// TwinCAT 3 PLC project PlcHammer
// Title: PlcHammer
// Company: TcOpenGroup
// ProjectVersion: 0.0.0.1
// ProgramVersion: 3.1.4023.0
// libraries:
//   Tc2_Math, * (Beckhoff Automation GmbH)
//   Tc2_Standard, * (Beckhoff Automation GmbH)
//   Tc2_System, * (Beckhoff Automation GmbH)
//   Tc3_Module, * (Beckhoff Automation GmbH)
//   TcoCore, 0.4.2.535 (Vortex.Library)
//   TcoData, 0.4.2.535 (Vortex.Library)
//   TcoDrivesBeckhoff, 0.4.2.535 (Vortex.Library)
//   TcoElements, 0.4.2.535 (Vortex.Library)
//   TcoIoBeckhoff, 0.4.2.535 (Vortex.Library)
//   TcoPneumatics, 0.4.2.535 (Vortex.Library)
// project tree:
//   Components/Drive/ DriveSim.TcPOU (not stored), DriveSimMoveAbsoluteTask.TcPOU (not stored), IDrive.TcIO (not stored)
//   Misc/Checkers/ Checkers.TcPOU (not stored), AnalogueValueCheck.TcDUT (not stored), eCheckResult.TcDUT (not stored)
//   / PlcTask.TcTTO (not stored)
//   POUs/ AppContext.TcPOU (not stored), TECH_MAIN.TcPOU
//   POUs/Data/ ProcessDataManager.TcPOU (not stored), RealValueSimulation.TcPOU (not stored), TechnologicalDataManager.TcPOU (not stored)
//   POUs/Data/Task Test mit Interlocking/ SubRoutine.TcPOU (not stored), SubRoutineAutoMode.TcPOU (not stored)
//   POUs/Station001/ Station001_Swift.TcPOU (not stored), IO.TcGVL (not stored), Station001.TcPOU, Station001_Components.TcPOU (not stored), Station001_GroundMode.TcPOU, Station001_AutomatMode.TcPOU (not stored), Station001_ProductionData.TcDUT, Station001_TechnologicalSettings.TcDUT (not stored)
// real-time tasks:
//   TASK PlcTask: cycle T#10ms, priority 20, ADS port 350
// motion (NC):
//   TASK NC-Task 1 SAF: cycle T#2ms, priority 4, ADS port 501
//   TASK NC-Task 1 SVB: cycle T#10ms, priority 8, ADS port 511
//   AXIS Axis 1 (id 1)
//     OtherSettings: AllowMotionCmdToSlave=true
//     encoder EncType=1
//     drive DrvType=5
//       Analog: TorqueSetpointScale=10, ScaleFactorActTorque=0.1
//       TimeComp: TaskDelayCycles=1
//     controller CtrType=1
//       CtrPara: PriorControlFactor=1
//         Observer: BandWidth=20
// variable links:
//   PlcHammer/PlcHammer Instance <-> NC-Task 1 SAF/Axes/Axis 1
//     PlcTask Inputs/IO.Axis1.NcToPlc <-> Outputs/ToPlc
//     PlcTask Outputs/IO.Axis1.PlcToNc <-> Inputs/FromPlc

// ---- POUs/Station001/Station001_ProductionData.TcDUT
TYPE Station001_ProductionData EXTENDS TcoData.Entity:
STRUCT
	DimX : AnalogueValueCheck;
	DimY : AnalogueValueCheck;
	DimZ : AnalogueValueCheck;
END_STRUCT
END_TYPE

// ---- POUs/TECH_MAIN.TcPOU
PROGRAM TECH_MAIN
VAR
	_app : AppContext;
	Alberts : AlbertsContext;
END_VAR

_app.Run();
_app.RtcSynchronize(TRUE, '', 60);
Alberts.Run();
Alberts.RtcSynchronize(TRUE,'',60);

END_PROGRAM

// ---- POUs/Station001/Station001.TcPOU
FUNCTION_BLOCK Station001 EXTENDS TcoCore.TcoObject 
VAR
	_components : Station001_Components(THIS^);
	
	_groundMode : Station001_GroundMode(THIS^, eRestoreMode.None);
	_automatMode : Station001_AutomatMode(THIS^, eRestoreMode.None);
	_swiftSequence   : Station001_Swift(THIS^, eRestoreMode.None);
	
	_groundModeTask : TcoCore.TcoTask(THIS^);
	_automatModeTask : TcoCore.TcoTask(THIS^);
	_serviceModeTask : TcoCore.TcoTask(THIS^);
	_swiftModeTask : TcoCore.TcoTask(THIS^);
	
	
	_processRecipies : ProcessDataManager(THIS^); 
    _processTraceabilty : ProcessDataManager(THIS^);
	_technologicalDataManager : TechnologicalDataManager(THIS^);
	
	_checkers : Checkers(THIS^);
END_VAR

_components();
_processRecipies();
_processTraceabilty();
_technologicalDataManager();


ServiceMode();
GroundMode();
AutomatMode();


IF(_swiftModeTask.Execute()) THEN
	Messenger.Trace('Service mode active');	
	_automatModeTask.Restore();
	_groundModeTask.Restore();
	_groundMode.Restore();
	_automatMode.Restore();
	_serviceModeTask.Restore();
	_swiftSequence.Run();
END_IF

METHOD AutomatMode : BOOL
VAR_INPUT
END_VAR
_automatModeTask.Enabled := _groundModeTask.Done;

IF(_automatModeTask.Execute()) THEN
	Messenger.Trace('Automat mode active');
	_serviceModeTask.Abort();
	_automatMode.Run();
END_IF
END_METHOD

PROPERTY Checkers : REFERENCE TO Checkers
GET
Checkers REF= _checkers;
END_GET
END_PROPERTY

PROPERTY Components : REFERENCE TO Station001_Components
GET
Components REF= _components;
END_GET
END_PROPERTY

PROPERTY ComponentsFeederTag : reference to FeederTags_Components
GET
ComponentsFeederTag ref= _componentsFeederTag;
END_GET
END_PROPERTY

METHOD GroundMode : BOOL
VAR_INPUT
END_VAR
IF(_groundModeTask.Execute()) THEN
	Messenger.Trace('Ground position mode active');
	_serviceModeTask.Restore();
	_automatModeTask.Restore();
	_automatMode.Restore();
	_groundMode.Run();
	_groundModeTask.DoneWhen(_groundMode.CurrentStep.ID = 300);
	IF _groundModeTask.Done THEN
		_groundMode.Restore();
	END_IF
END_IF
END_METHOD

PROPERTY ProcessRecepie : REFERENCE TO ProcessDataManager
GET
ProcessRecepie REF= _processRecipies;
END_GET
END_PROPERTY

PROPERTY ProcessTraceabilty : REFERENCE TO ProcessDataManager
GET
ProcessTraceabilty REF= _processTraceabilty;
END_GET
END_PROPERTY

PROPERTY  ProductionData : REFERENCE TO Station001_ProductionData
GET
ProductionData REF= _processTraceabilty._data;
END_GET
END_PROPERTY

METHOD ServiceMode
VAR_INPUT
END_VAR
IF(_serviceModeTask.Execute()) THEN
	Messenger.Trace('Service mode active');	
	_automatModeTask.Restore();
	_groundModeTask.Restore();
	_groundMode.Restore();
	_automatMode.Restore();
	_components.Service();
END_IF
END_METHOD

PROPERTY TechnologicalDataManager : REFERENCE TO TechnologicalDataManager
GET
TechnologicalDataManager REF= _technologicalDataManager;
END_GET
END_PROPERTY

END_FUNCTION_BLOCK

// ---- POUs/Station001/Station001_GroundMode.TcPOU
FUNCTION_BLOCK Station001_GroundMode EXTENDS TcoCore.TcoSequencer

METHOD InvokeSubSeqB : BOOL
VAR_INPUT
END_VAR
_subRoutineA_AutomatModeTask.Invoke();
END_METHOD

(*~
	<docu>
		<summary>
			Main method of the sequener. Custom code needs to be placed here. The sequencer is executed by call of InstanceName.Run() method.
			This method is abstract, and it must be overridden in derived block.
		</summary>
	</docu>
~*)
METHOD PROTECTED  Main : BOOL
VAR CONSTANT
	HORIZONTAL_AXIS_HOME_POSITION : LREAL := 0.0;
END_VAR
IF (Step(10, TRUE, 'RESTORE ALL COMPONENTS')) THEN
    //--------------------------------------------
	Station.Components._horizontalNcAxis.Restore();
	Station.Components._verticalPiston.Restore();
	Station.Components._gripperPiston.Restore();
    StepCompleteWhen(TRUE);
    //--------------------------------------------	
END_IF;

IF (Step(100, TRUE, 'MOVE VERTICAL AXIS UP')) THEN
    //--------------------------------------------
    StepCompleteWhen(Station.Components.VerticalAxis.MoveToHome().Done);
    //--------------------------------------------	
END_IF;

IF (Step(125, TRUE, 'LOAD TECHNOLOGICAL SETTINGS')) THEN
    //--------------------------------------------
    StepCompleteWhen(Station.TechnologicalDataManager.Read('default').Done);
    //--------------------------------------------	
END_IF;

IF (Step(150, NOT Station.Components.HorizontalNcAxis.DriveRef._axisStatus.Homed, 'HORIZONTAL AXIS HOMING')) THEN
    //--------------------------------------------
    StepCompleteWhen(Station.Components.HorizontalNcAxis.DriveRef.Home(inPosition := 0,
            inHomingMode := TcoDrivesBeckhoff.eHomingMode.MC_Direct,
            inClearPositionLag := FALSE,
            inSearchDirection := TcoDrivesBeckhoff.eDirection.MC_Undefined_Direction,
            inSearchVelocity := 100.0,
            inSyncDirection := TcoDrivesBeckhoff.eDirection.MC_Undefined_Direction,
            inSyncVelocity := 100.0,
            inReferenceMode := TcoDrivesBeckhoff.eEncoderReferenceMode.ENCODERREFERENCEMODE_DEFAULT).Done);
    //--------------------------------------------	
END_IF;

IF (Step(200, TRUE, 'MOVE HORIZONTAL AXIS TO BASE POSITION & OPEN GRIPPER')) THEN
    //--------------------------------------------
    IF (Station.Components.HorizontalNcAxis.DriveRef.MoveAbsolute(HORIZONTAL_AXIS_HOME_POSITION,
        THIS^.Station.TechnologicalDataManager._data.AxisSpeed,
        THIS^.Station.TechnologicalDataManager._data.AxisAcc,
        THIS^.Station.TechnologicalDataManager._data.AxisDcc,
        THIS^.Station.TechnologicalDataManager._data.AxisJerk).Done AND
        Station.Components.Gripper.MoveToHome().Done) THEN
        CompleteStep();
    END_IF;
    //--------------------------------------------	
END_IF;

IF (Step(300, TRUE, 'GROUND POSITION DONE')) THEN
    //--------------------------------------------
    ;
    //--------------------------------------------	
END_IF;
END_METHOD

(*~
	<docu>
		<summary>
			This method is executed upon step completion.
			This method can be overridden in derived block by custom logic.
		</summary>			
	</docu>	
~*)
METHOD PROTECTED OnStepCompleted
END_METHOD

PROPERTY Station : REFERENCE TO Station001
GET
VAR
    _station : POINTER TO Station001;
END_VAR
IF __QUERYPOINTER(_Parent,_station) THEN // Check if _Parent is Station001
	Station REF= _station^;              // If the check is successful dereference a pointer. simlar to THIS^ or SUPER^
END_IF
END_GET
END_PROPERTY

METHOD SubSeqA_AutoMode : bool
VAR_INPUT
END_VAR
IF _subRoutineA_AutomatModeTask.Execute() THEN
    _subRoutineA_AutomatMode.Run();
    _subRoutineA_AutomatModeTask.DoneWhen(_subRoutineA_AutomatMode.CurrentStep.ID = 400);
    IF _subRoutineA_AutomatModeTask.Done THEN
        _subRoutineA_AutomatMode.Restore();
       
	END_IF
END_IF

SubSeqA_AutoMode:= _subRoutineA_AutomatModeTask.Done;
END_METHOD

END_FUNCTION_BLOCK
